Staubli VAL3: cmdSwitchOn.pgx

public program cmdSwitchOn(num& x_nAxNum)
begin
  //"switch on"设置为true
  doFaultReset[x_nAxNum]=false
  doEnableOp[x_nAxNum]=false
  doQuickStop[x_nAxNum]=true
  doEnableVoltage[x_nAxNum]=true
  doSwitchOn[x_nAxNum]=true
  delay(0.1)
end
